PROGRAM MAIN
VAR
	{attribute 'pytmc' := 'pv: TEST:NEODRY:01'}
	test : BOOL;
END_VAR

test_pump();

test_pump_2();

END_PROGRAM

(* stored: Version 1.1.0.1
   POU MAIN: Id {93f0cc46-ee06-47a7-bfaf-d9ed4a72d957}, SpecialFunc None *)
